// TIA Portal project "TestPID" (V16)

(* hardware
DEVICE "S7-1200 station_1"  S7-1200 Station
   slot 0: "Rack_0"  S7-1200 Rack  Rack  V1.0
   slot 1: "PLC_1"  CPU 1214C DC/DC/DC  6ES7 214-1AG40-0XB0  V4.4
*)

// ===== PLC "PLC_1"  CPU 1214C DC/DC/DC =====

VAR_GLOBAL   // PLC tag table "Default tag table"
   "set" AT %MD0 : Real;
   "in" AT %MD4 : Real;
   "out" AT %MD8 : Real;
   "Invert_Colder" AT %M12.0 : Bool;
   "PID_1_Reset" AT %M12.1 : Bool;
   "PID_Mode" AT %MW14 : Int;
END_VAR

FUNCTION_BLOCK "Block_1"   // FB1, SCL
{ S7_Optimized_Access := 'TRUE' }
VERSION : 0.1
BEGIN
END_FUNCTION_BLOCK

ORGANIZATION_BLOCK "Main"   // OB1, LAD, ProgramCycle
TITLE = "Main Program Sweep (Cycle)"
{ S7_Optimized_Access := 'TRUE' }
VERSION : 0.1
BEGIN

REGION Network 1
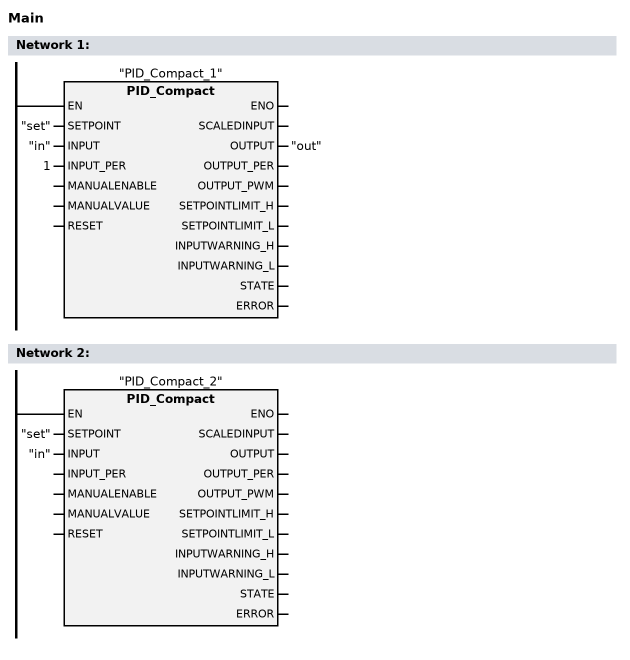
   "PID_Compact_1"(Setpoint := "set", Input := "in", Input_PER := 1, Output => "out");   // PID_Compact
END_REGION

REGION Network 2
   "PID_Compact_2"(Setpoint := "set", Input := "in");   // PID_Compact
END_REGION

REGION Network 3 (SCL)
   "PID_Compact_1".sPid_Cmpt.b_InvCtrl := "Invert_Colder";
   "PID_Compact_1".Reset := "PID_1_Reset";

   "PID_Mode" := "PID_Compact_1".sRet.i_Mode;
END_REGION
END_ORGANIZATION_BLOCK